Staubli VAL3: recvTrajPtCartesian.pgx

public program recvTrajPtCartesian(bool& x_bFlag)
begin
  // attempt to receive message ID 31 data (prefix and header are in rosGenericMsg)
  rosTrajPtCartesianMsg.prefix.nLength=rosGenericMsg.prefix.nLength
  rosTrajPtCartesianMsg.header.nMsgType=rosGenericMsg.header.nMsgType
  rosTrajPtCartesianMsg.header.nCommType=rosGenericMsg.header.nCommType
  rosTrajPtCartesianMsg.header.nReplyCode=rosGenericMsg.header.nReplyCode

  call recvData(siTcpIpMotion,rosTrajPtCartesianMsg.body.nData,nInConnFlag,x_bFlag)
end
